GLOBALCONSTANTS STATES (* Global constants *)
  (* Standard: 61499-1 *)
  (* Version 1.0, 2025-05-23, franz *)
  PACKAGE Verteiler::LinksRechts;
  VAR_GLOBAL CONSTANT
    Rechtslauf : STRING := STRING#'Rechtslauf';
    Linkslauf : STRING := STRING#'Linkslauf';
    Linkslauf_Pause : STRING := STRING#'Linkslauf_Pause';
    Rechtslauf_Pause : STRING := STRING#'Rechtslauf_Pause';
  END_VAR
END_GLOBALCONSTANTS
